{attribute 'GeneratedUsingTerminal: EL1918-0000-0016'}
{attribute addProperty BoxType "EL1918-0000-0016"}
{attribute addProperty Id "Safe_Logic_StateAT %I*USINT1Cycle_CounterAT %I*USINT1"}
{attribute addProperty CRC "4008261774"}
{attribute addProperty Size "2"}
TYPE FSLOGIC_Inputs_EEE9388E EXTENDS InputBase_8311D824 :
STRUCT
	{attribute addProperty Name "Safe_Logic_State"}
	Safe_Logic_State AT %I* : USINT;
	{attribute addProperty Name "Cycle_Counter"}
	Cycle_Counter AT %I* : USINT;
END_STRUCT
END_TYPE

(* stored: Version 1.2.0.0, ProductVersion 3.1.4024.11
   DUT FSLOGIC_Inputs_EEE9388E: Id {996d10d4-54f4-4e2c-a1e6-6b58d8888666} *)
